FUNCTION_BLOCK "FB33 Ausgaege an FG"	// FB 33
TITLE = Ausgänge für Farbgrafik in Datenworte des DB33 speichern
//Erstellung:
//Datum        Bearbeiter                                                 Version
//--------------------------------------------------------------------------------
//00.00.00     xxx                                                        01.00.00
//
//Änderungen:
//Nr. Datum    Bearb Beschreibung                                   Marke Version
//--------------------------------------------------------------------------------
//01  00.00.00                                                      (xxx) xx.xx.xx
//
//--------------------------------------------------------------------------------
//
//
AUTHOR : sra
FAMILY : SCADA
NAME : outputs
VERSION : 0.0
VAR
  output_0_0 : BOOL ;
  output_0_1 : BOOL ;
  output_0_2 : BOOL ;
  output_0_3 : BOOL ;
  output_0_4 : BOOL ;
  output_0_5 : BOOL ;
  output_0_6 : BOOL ;
  output_0_7 : BOOL ;
  output_1_0 : BOOL ;
  output_1_1 : BOOL ;
  output_1_2 : BOOL ;
  output_1_3 : BOOL ;
  output_1_4 : BOOL ;
  output_1_5 : BOOL ;
  output_1_6 : BOOL ;
  output_1_7 : BOOL ;
  output_2_0 : BOOL ;
  output_2_1 : BOOL ;
  output_2_2 : BOOL ;
  output_2_3 : BOOL ;
  output_2_4 : BOOL ;
  output_2_5 : BOOL ;
  output_2_6 : BOOL ;
  output_2_7 : BOOL ;
  output_3_0 : BOOL ;
  output_3_1 : BOOL ;
  output_3_2 : BOOL ;
  output_3_3 : BOOL ;
  output_3_4 : BOOL ;
  output_3_5 : BOOL ;
  output_3_6 : BOOL ;
  output_3_7 : BOOL ;
  output_4_0 : BOOL ;
  output_4_1 : BOOL ;
  output_4_2 : BOOL ;
  output_4_3 : BOOL ;
  output_4_4 : BOOL ;
  output_4_5 : BOOL ;
  output_4_6 : BOOL ;
  output_4_7 : BOOL ;
  output_5_0 : BOOL ;
  output_5_1 : BOOL ;
  output_5_2 : BOOL ;
  output_5_3 : BOOL ;
  output_5_4 : BOOL ;
  output_5_5 : BOOL ;
  output_5_6 : BOOL ;
  output_5_7 : BOOL ;
  output_6_0 : BOOL ;
  output_6_1 : BOOL ;
  output_6_2 : BOOL ;
  output_6_3 : BOOL ;
  output_6_4 : BOOL ;
  output_6_5 : BOOL ;
  output_6_6 : BOOL ;
  output_6_7 : BOOL ;
  output_7_0 : BOOL ;
  output_7_1 : BOOL ;
  output_7_2 : BOOL ;
  output_7_3 : BOOL ;
  output_7_4 : BOOL ;
  output_7_5 : BOOL ;
  output_7_6 : BOOL ;
  output_7_7 : BOOL ;
  output_8_0 : BOOL ;
  output_8_1 : BOOL ;
  output_8_2 : BOOL ;
  output_8_3 : BOOL ;
  output_8_4 : BOOL ;
  output_8_5 : BOOL ;
  output_8_6 : BOOL ;
  output_8_7 : BOOL ;
  output_9_0 : BOOL ;
  output_9_1 : BOOL ;
  output_9_2 : BOOL ;
  output_9_3 : BOOL ;
  output_9_4 : BOOL ;
  output_9_5 : BOOL ;
  output_9_6 : BOOL ;
  output_9_7 : BOOL ;
  output_10_0 : BOOL ;
  output_10_1 : BOOL ;
  output_10_2 : BOOL ;
  output_10_3 : BOOL ;
  output_10_4 : BOOL ;
  output_10_5 : BOOL ;
  output_10_6 : BOOL ;
  output_10_7 : BOOL ;
  output_11_0 : BOOL ;
  output_11_1 : BOOL ;
  output_11_2 : BOOL ;
  output_11_3 : BOOL ;
  output_11_4 : BOOL ;
  output_11_5 : BOOL ;
  output_11_6 : BOOL ;
  output_11_7 : BOOL ;
  output_12_0 : BOOL ;
  output_12_1 : BOOL ;
  output_12_2 : BOOL ;
  output_12_3 : BOOL ;
  output_12_4 : BOOL ;
  output_12_5 : BOOL ;
  output_12_6 : BOOL ;
  output_12_7 : BOOL ;
  output_13_0 : BOOL ;
  output_13_1 : BOOL ;
  output_13_2 : BOOL ;
  output_13_3 : BOOL ;
  output_13_4 : BOOL ;
  output_13_5 : BOOL ;
  output_13_6 : BOOL ;
  output_13_7 : BOOL ;
  output_14_0 : BOOL ;
  output_14_1 : BOOL ;
  output_14_2 : BOOL ;
  output_14_3 : BOOL ;
  output_14_4 : BOOL ;
  output_14_5 : BOOL ;
  output_14_6 : BOOL ;
  output_14_7 : BOOL ;
  output_15_0 : BOOL ;
  output_15_1 : BOOL ;
  output_15_2 : BOOL ;
  output_15_3 : BOOL ;
  output_15_4 : BOOL ;
  output_15_5 : BOOL ;
  output_15_6 : BOOL ;
  output_15_7 : BOOL ;
  output_16_0 : BOOL ;
  output_16_1 : BOOL ;
  output_16_2 : BOOL ;
  output_16_3 : BOOL ;
  output_16_4 : BOOL ;
  output_16_5 : BOOL ;
  output_16_6 : BOOL ;
  output_16_7 : BOOL ;
  output_17_0 : BOOL ;
  output_17_1 : BOOL ;
  output_17_2 : BOOL ;
  output_17_3 : BOOL ;
  output_17_4 : BOOL ;
  output_17_5 : BOOL ;
  output_17_6 : BOOL ;
  output_17_7 : BOOL ;
  output_18_0 : BOOL ;
  output_18_1 : BOOL ;
  output_18_2 : BOOL ;
  output_18_3 : BOOL ;
  output_18_4 : BOOL ;
  output_18_5 : BOOL ;
  output_18_6 : BOOL ;
  output_18_7 : BOOL ;
  output_19_0 : BOOL ;
  output_19_1 : BOOL ;
  output_19_2 : BOOL ;
  output_19_3 : BOOL ;
  output_19_4 : BOOL ;
  output_19_5 : BOOL ;
  output_19_6 : BOOL ;
  output_19_7 : BOOL ;
  output_20_0 : BOOL ;
  output_20_1 : BOOL ;
  output_20_2 : BOOL ;
  output_20_3 : BOOL ;
  output_20_4 : BOOL ;
  output_20_5 : BOOL ;
  output_20_6 : BOOL ;
  output_20_7 : BOOL ;
  output_21_0 : BOOL ;
  output_21_1 : BOOL ;
  output_21_2 : BOOL ;
  output_21_3 : BOOL ;
  output_21_4 : BOOL ;
  output_21_5 : BOOL ;
  output_21_6 : BOOL ;
  output_21_7 : BOOL ;
  output_22_0 : BOOL ;
  output_22_1 : BOOL ;
  output_22_2 : BOOL ;
  output_22_3 : BOOL ;
  output_22_4 : BOOL ;
  output_22_5 : BOOL ;
  output_22_6 : BOOL ;
  output_22_7 : BOOL ;
  output_23_0 : BOOL ;
  output_23_1 : BOOL ;
  output_23_2 : BOOL ;
  output_23_3 : BOOL ;
  output_23_4 : BOOL ;
  output_23_5 : BOOL ;
  output_23_6 : BOOL ;
  output_23_7 : BOOL ;
  output_24_0 : BOOL ;
  output_24_1 : BOOL ;
  output_24_2 : BOOL ;
  output_24_3 : BOOL ;
  output_24_4 : BOOL ;
  output_24_5 : BOOL ;
  output_24_6 : BOOL ;
  output_24_7 : BOOL ;
  output_25_0 : BOOL ;
  output_25_1 : BOOL ;
  output_25_2 : BOOL ;
  output_25_3 : BOOL ;
  output_25_4 : BOOL ;
  output_25_5 : BOOL ;
  output_25_6 : BOOL ;
  output_25_7 : BOOL ;
  output_26_0 : BOOL ;
  output_26_1 : BOOL ;
  output_26_2 : BOOL ;
  output_26_3 : BOOL ;
  output_26_4 : BOOL ;
  output_26_5 : BOOL ;
  output_26_6 : BOOL ;
  output_26_7 : BOOL ;
  output_27_0 : BOOL ;
  output_27_1 : BOOL ;
  output_27_2 : BOOL ;
  output_27_3 : BOOL ;
  output_27_4 : BOOL ;
  output_27_5 : BOOL ;
  output_27_6 : BOOL ;
  output_27_7 : BOOL ;
  output_28_0 : BOOL ;
  output_28_1 : BOOL ;
  output_28_2 : BOOL ;
  output_28_3 : BOOL ;
  output_28_4 : BOOL ;
  output_28_5 : BOOL ;
  output_28_6 : BOOL ;
  output_28_7 : BOOL ;
  output_29_0 : BOOL ;
  output_29_1 : BOOL ;
  output_29_2 : BOOL ;
  output_29_3 : BOOL ;
  output_29_4 : BOOL ;
  output_29_5 : BOOL ;
  output_29_6 : BOOL ;
  output_29_7 : BOOL ;
  output_30_0 : BOOL ;
  output_30_1 : BOOL ;
  output_30_2 : BOOL ;
  output_30_3 : BOOL ;
  output_30_4 : BOOL ;
  output_30_5 : BOOL ;
  output_30_6 : BOOL ;
  output_30_7 : BOOL ;
  output_31_0 : BOOL ;
  output_31_1 : BOOL ;
  output_31_2 : BOOL ;
  output_31_3 : BOOL ;
  output_31_4 : BOOL ;
  output_31_5 : BOOL ;
  output_31_6 : BOOL ;
  output_31_7 : BOOL ;
  output_32_0 : BOOL ;
  output_32_1 : BOOL ;
  output_32_2 : BOOL ;
  output_32_3 : BOOL ;
  output_32_4 : BOOL ;
  output_32_5 : BOOL ;
  output_32_6 : BOOL ;
  output_32_7 : BOOL ;
  output_33_0 : BOOL ;
  output_33_1 : BOOL ;
  output_33_2 : BOOL ;
  output_33_3 : BOOL ;
  output_33_4 : BOOL ;
  output_33_5 : BOOL ;
  output_33_6 : BOOL ;
  output_33_7 : BOOL ;
  output_34_0 : BOOL ;
  output_34_1 : BOOL ;
  output_34_2 : BOOL ;
  output_34_3 : BOOL ;
  output_34_4 : BOOL ;
  output_34_5 : BOOL ;
  output_34_6 : BOOL ;
  output_34_7 : BOOL ;
  output_35_0 : BOOL ;
  output_35_1 : BOOL ;
  output_35_2 : BOOL ;
  output_35_3 : BOOL ;
  output_35_4 : BOOL ;
  output_35_5 : BOOL ;
  output_35_6 : BOOL ;
  output_35_7 : BOOL ;
  output_36_0 : BOOL ;
  output_36_1 : BOOL ;
  output_36_2 : BOOL ;
  output_36_3 : BOOL ;
  output_36_4 : BOOL ;
  output_36_5 : BOOL ;
  output_36_6 : BOOL ;
  output_36_7 : BOOL ;
  output_37_0 : BOOL ;
  output_37_1 : BOOL ;
  output_37_2 : BOOL ;
  output_37_3 : BOOL ;
  output_37_4 : BOOL ;
  output_37_5 : BOOL ;
  output_37_6 : BOOL ;
  output_37_7 : BOOL ;
  output_38_0 : BOOL ;
  output_38_1 : BOOL ;
  output_38_2 : BOOL ;
  output_38_3 : BOOL ;
  output_38_4 : BOOL ;
  output_38_5 : BOOL ;
  output_38_6 : BOOL ;
  output_38_7 : BOOL ;
  output_39_0 : BOOL ;
  output_39_1 : BOOL ;
  output_39_2 : BOOL ;
  output_39_3 : BOOL ;
  output_39_4 : BOOL ;
  output_39_5 : BOOL ;
  output_39_6 : BOOL ;
  output_39_7 : BOOL ;
  output_40_0 : BOOL ;
  output_40_1 : BOOL ;
  output_40_2 : BOOL ;
  output_40_3 : BOOL ;
  output_40_4 : BOOL ;
  output_40_5 : BOOL ;
  output_40_6 : BOOL ;
  output_40_7 : BOOL ;
  output_41_0 : BOOL ;
  output_41_1 : BOOL ;
  output_41_2 : BOOL ;
  output_41_3 : BOOL ;
  output_41_4 : BOOL ;
  output_41_5 : BOOL ;
  output_41_6 : BOOL ;
  output_41_7 : BOOL ;
  output_42_0 : BOOL ;
  output_42_1 : BOOL ;
  output_42_2 : BOOL ;
  output_42_3 : BOOL ;
  output_42_4 : BOOL ;
  output_42_5 : BOOL ;
  output_42_6 : BOOL ;
  output_42_7 : BOOL ;
  output_43_0 : BOOL ;
  output_43_1 : BOOL ;
  output_43_2 : BOOL ;
  output_43_3 : BOOL ;
  output_43_4 : BOOL ;
  output_43_5 : BOOL ;
  output_43_6 : BOOL ;
  output_43_7 : BOOL ;
  output_44_0 : BOOL ;
  output_44_1 : BOOL ;
  output_44_2 : BOOL ;
  output_44_3 : BOOL ;
  output_44_4 : BOOL ;
  output_44_5 : BOOL ;
  output_44_6 : BOOL ;
  output_44_7 : BOOL ;
  output_45_0 : BOOL ;
  output_45_1 : BOOL ;
  output_45_2 : BOOL ;
  output_45_3 : BOOL ;
  output_45_4 : BOOL ;
  output_45_5 : BOOL ;
  output_45_6 : BOOL ;
  output_45_7 : BOOL ;
  output_46_0 : BOOL ;
  output_46_1 : BOOL ;
  output_46_2 : BOOL ;
  output_46_3 : BOOL ;
  output_46_4 : BOOL ;
  output_46_5 : BOOL ;
  output_46_6 : BOOL ;
  output_46_7 : BOOL ;
  output_47_0 : BOOL ;
  output_47_1 : BOOL ;
  output_47_2 : BOOL ;
  output_47_3 : BOOL ;
  output_47_4 : BOOL ;
  output_47_5 : BOOL ;
  output_47_6 : BOOL ;
  output_47_7 : BOOL ;
  output_48_0 : BOOL ;
  output_48_1 : BOOL ;
  output_48_2 : BOOL ;
  output_48_3 : BOOL ;
  output_48_4 : BOOL ;
  output_48_5 : BOOL ;
  output_48_6 : BOOL ;
  output_48_7 : BOOL ;
  output_49_0 : BOOL ;
  output_49_1 : BOOL ;
  output_49_2 : BOOL ;
  output_49_3 : BOOL ;
  output_49_4 : BOOL ;
  output_49_5 : BOOL ;
  output_49_6 : BOOL ;
  output_49_7 : BOOL ;
  output_50_0 : BOOL ;
  output_50_1 : BOOL ;
  output_50_2 : BOOL ;
  output_50_3 : BOOL ;
  output_50_4 : BOOL ;
  output_50_5 : BOOL ;
  output_50_6 : BOOL ;
  output_50_7 : BOOL ;
  output_51_0 : BOOL ;
  output_51_1 : BOOL ;
  output_51_2 : BOOL ;
  output_51_3 : BOOL ;
  output_51_4 : BOOL ;
  output_51_5 : BOOL ;
  output_51_6 : BOOL ;
  output_51_7 : BOOL ;
  output_52_0 : BOOL ;
  output_52_1 : BOOL ;
  output_52_2 : BOOL ;
  output_52_3 : BOOL ;
  output_52_4 : BOOL ;
  output_52_5 : BOOL ;
  output_52_6 : BOOL ;
  output_52_7 : BOOL ;
  output_53_0 : BOOL ;
  output_53_1 : BOOL ;
  output_53_2 : BOOL ;
  output_53_3 : BOOL ;
  output_53_4 : BOOL ;
  output_53_5 : BOOL ;
  output_53_6 : BOOL ;
  output_53_7 : BOOL ;
  output_54_0 : BOOL ;
  output_54_1 : BOOL ;
  output_54_2 : BOOL ;
  output_54_3 : BOOL ;
  output_54_4 : BOOL ;
  output_54_5 : BOOL ;
  output_54_6 : BOOL ;
  output_54_7 : BOOL ;
  output_55_0 : BOOL ;
  output_55_1 : BOOL ;
  output_55_2 : BOOL ;
  output_55_3 : BOOL ;
  output_55_4 : BOOL ;
  output_55_5 : BOOL ;
  output_55_6 : BOOL ;
  output_55_7 : BOOL ;
  output_56_0 : BOOL ;
  output_56_1 : BOOL ;
  output_56_2 : BOOL ;
  output_56_3 : BOOL ;
  output_56_4 : BOOL ;
  output_56_5 : BOOL ;
  output_56_6 : BOOL ;
  output_56_7 : BOOL ;
  output_57_0 : BOOL ;
  output_57_1 : BOOL ;
  output_57_2 : BOOL ;
  output_57_3 : BOOL ;
  output_57_4 : BOOL ;
  output_57_5 : BOOL ;
  output_57_6 : BOOL ;
  output_57_7 : BOOL ;
  output_58_0 : BOOL ;
  output_58_1 : BOOL ;
  output_58_2 : BOOL ;
  output_58_3 : BOOL ;
  output_58_4 : BOOL ;
  output_58_5 : BOOL ;
  output_58_6 : BOOL ;
  output_58_7 : BOOL ;
  output_59_0 : BOOL ;
  output_59_1 : BOOL ;
  output_59_2 : BOOL ;
  output_59_3 : BOOL ;
  output_59_4 : BOOL ;
  output_59_5 : BOOL ;
  output_59_6 : BOOL ;
  output_59_7 : BOOL ;
  output_60_0 : BOOL ;
  output_60_1 : BOOL ;
  output_60_2 : BOOL ;
  output_60_3 : BOOL ;
  output_60_4 : BOOL ;
  output_60_5 : BOOL ;
  output_60_6 : BOOL ;
  output_60_7 : BOOL ;
  output_61_0 : BOOL ;
  output_61_1 : BOOL ;
  output_61_2 : BOOL ;
  output_61_3 : BOOL ;
  output_61_4 : BOOL ;
  output_61_5 : BOOL ;
  output_61_6 : BOOL ;
  output_61_7 : BOOL ;
  output_62_0 : BOOL ;
  output_62_1 : BOOL ;
  output_62_2 : BOOL ;
  output_62_3 : BOOL ;
  output_62_4 : BOOL ;
  output_62_5 : BOOL ;
  output_62_6 : BOOL ;
  output_62_7 : BOOL ;
  output_63_0 : BOOL ;
  output_63_1 : BOOL ;
  output_63_2 : BOOL ;
  output_63_3 : BOOL ;
  output_63_4 : BOOL ;
  output_63_5 : BOOL ;
  output_63_6 : BOOL ;
  output_63_7 : BOOL ;
  output_64_0 : BOOL ;
  output_64_1 : BOOL ;
  output_64_2 : BOOL ;
  output_64_3 : BOOL ;
  output_64_4 : BOOL ;
  output_64_5 : BOOL ;
  output_64_6 : BOOL ;
  output_64_7 : BOOL ;
  output_65_0 : BOOL ;
  output_65_1 : BOOL ;
  output_65_2 : BOOL ;
  output_65_3 : BOOL ;
  output_65_4 : BOOL ;
  output_65_5 : BOOL ;
  output_65_6 : BOOL ;
  output_65_7 : BOOL ;
  output_66_0 : BOOL ;
  output_66_1 : BOOL ;
  output_66_2 : BOOL ;
  output_66_3 : BOOL ;
  output_66_4 : BOOL ;
  output_66_5 : BOOL ;
  output_66_6 : BOOL ;
  output_66_7 : BOOL ;
  output_67_0 : BOOL ;
  output_67_1 : BOOL ;
  output_67_2 : BOOL ;
  output_67_3 : BOOL ;
  output_67_4 : BOOL ;
  output_67_5 : BOOL ;
  output_67_6 : BOOL ;
  output_67_7 : BOOL ;
  output_68_0 : BOOL ;
  output_68_1 : BOOL ;
  output_68_2 : BOOL ;
  output_68_3 : BOOL ;
  output_68_4 : BOOL ;
  output_68_5 : BOOL ;
  output_68_6 : BOOL ;
  output_68_7 : BOOL ;
  output_69_0 : BOOL ;
  output_69_1 : BOOL ;
  output_69_2 : BOOL ;
  output_69_3 : BOOL ;
  output_69_4 : BOOL ;
  output_69_5 : BOOL ;
  output_69_6 : BOOL ;
  output_69_7 : BOOL ;
  output_70_0 : BOOL ;
  output_70_1 : BOOL ;
  output_70_2 : BOOL ;
  output_70_3 : BOOL ;
  output_70_4 : BOOL ;
  output_70_5 : BOOL ;
  output_70_6 : BOOL ;
  output_70_7 : BOOL ;
  output_71_0 : BOOL ;
  output_71_1 : BOOL ;
  output_71_2 : BOOL ;
  output_71_3 : BOOL ;
  output_71_4 : BOOL ;
  output_71_5 : BOOL ;
  output_71_6 : BOOL ;
  output_71_7 : BOOL ;
  output_72_0 : BOOL ;
  output_72_1 : BOOL ;
  output_72_2 : BOOL ;
  output_72_3 : BOOL ;
  output_72_4 : BOOL ;
  output_72_5 : BOOL ;
  output_72_6 : BOOL ;
  output_72_7 : BOOL ;
  output_73_0 : BOOL ;
  output_73_1 : BOOL ;
  output_73_2 : BOOL ;
  output_73_3 : BOOL ;
  output_73_4 : BOOL ;
  output_73_5 : BOOL ;
  output_73_6 : BOOL ;
  output_73_7 : BOOL ;
  output_74_0 : BOOL ;
  output_74_1 : BOOL ;
  output_74_2 : BOOL ;
  output_74_3 : BOOL ;
  output_74_4 : BOOL ;
  output_74_5 : BOOL ;
  output_74_6 : BOOL ;
  output_74_7 : BOOL ;
  output_75_0 : BOOL ;
  output_75_1 : BOOL ;
  output_75_2 : BOOL ;
  output_75_3 : BOOL ;
  output_75_4 : BOOL ;
  output_75_5 : BOOL ;
  output_75_6 : BOOL ;
  output_75_7 : BOOL ;
  output_76_0 : BOOL ;
  output_76_1 : BOOL ;
  output_76_2 : BOOL ;
  output_76_3 : BOOL ;
  output_76_4 : BOOL ;
  output_76_5 : BOOL ;
  output_76_6 : BOOL ;
  output_76_7 : BOOL ;
  output_77_0 : BOOL ;
  output_77_1 : BOOL ;
  output_77_2 : BOOL ;
  output_77_3 : BOOL ;
  output_77_4 : BOOL ;
  output_77_5 : BOOL ;
  output_77_6 : BOOL ;
  output_77_7 : BOOL ;
  output_78_0 : BOOL ;
  output_78_1 : BOOL ;
  output_78_2 : BOOL ;
  output_78_3 : BOOL ;
  output_78_4 : BOOL ;
  output_78_5 : BOOL ;
  output_78_6 : BOOL ;
  output_78_7 : BOOL ;
  output_79_0 : BOOL ;
  output_79_1 : BOOL ;
  output_79_2 : BOOL ;
  output_79_3 : BOOL ;
  output_79_4 : BOOL ;
  output_79_5 : BOOL ;
  output_79_6 : BOOL ;
  output_79_7 : BOOL ;
  output_80_0 : BOOL ;
  output_80_1 : BOOL ;
  output_80_2 : BOOL ;
  output_80_3 : BOOL ;
  output_80_4 : BOOL ;
  output_80_5 : BOOL ;
  output_80_6 : BOOL ;
  output_80_7 : BOOL ;
  output_81_0 : BOOL ;
  output_81_1 : BOOL ;
  output_81_2 : BOOL ;
  output_81_3 : BOOL ;
  output_81_4 : BOOL ;
  output_81_5 : BOOL ;
  output_81_6 : BOOL ;
  output_81_7 : BOOL ;
  output_82_0 : BOOL ;
  output_82_1 : BOOL ;
  output_82_2 : BOOL ;
  output_82_3 : BOOL ;
  output_82_4 : BOOL ;
  output_82_5 : BOOL ;
  output_82_6 : BOOL ;
  output_82_7 : BOOL ;
  output_83_0 : BOOL ;
  output_83_1 : BOOL ;
  output_83_2 : BOOL ;
  output_83_3 : BOOL ;
  output_83_4 : BOOL ;
  output_83_5 : BOOL ;
  output_83_6 : BOOL ;
  output_83_7 : BOOL ;
  output_84_0 : BOOL ;
  output_84_1 : BOOL ;
  output_84_2 : BOOL ;
  output_84_3 : BOOL ;
  output_84_4 : BOOL ;
  output_84_5 : BOOL ;
  output_84_6 : BOOL ;
  output_84_7 : BOOL ;
  output_85_0 : BOOL ;
  output_85_1 : BOOL ;
  output_85_2 : BOOL ;
  output_85_3 : BOOL ;
  output_85_4 : BOOL ;
  output_85_5 : BOOL ;
  output_85_6 : BOOL ;
  output_85_7 : BOOL ;
  output_86_0 : BOOL ;
  output_86_1 : BOOL ;
  output_86_2 : BOOL ;
  output_86_3 : BOOL ;
  output_86_4 : BOOL ;
  output_86_5 : BOOL ;
  output_86_6 : BOOL ;
  output_86_7 : BOOL ;
  output_87_0 : BOOL ;
  output_87_1 : BOOL ;
  output_87_2 : BOOL ;
  output_87_3 : BOOL ;
  output_87_4 : BOOL ;
  output_87_5 : BOOL ;
  output_87_6 : BOOL ;
  output_87_7 : BOOL ;
  output_88_0 : BOOL ;
  output_88_1 : BOOL ;
  output_88_2 : BOOL ;
  output_88_3 : BOOL ;
  output_88_4 : BOOL ;
  output_88_5 : BOOL ;
  output_88_6 : BOOL ;
  output_88_7 : BOOL ;
  output_89_0 : BOOL ;
  output_89_1 : BOOL ;
  output_89_2 : BOOL ;
  output_89_3 : BOOL ;
  output_89_4 : BOOL ;
  output_89_5 : BOOL ;
  output_89_6 : BOOL ;
  output_89_7 : BOOL ;
  output_90_0 : BOOL ;
  output_90_1 : BOOL ;
  output_90_2 : BOOL ;
  output_90_3 : BOOL ;
  output_90_4 : BOOL ;
  output_90_5 : BOOL ;
  output_90_6 : BOOL ;
  output_90_7 : BOOL ;
  output_91_0 : BOOL ;
  output_91_1 : BOOL ;
  output_91_2 : BOOL ;
  output_91_3 : BOOL ;
  output_91_4 : BOOL ;
  output_91_5 : BOOL ;
  output_91_6 : BOOL ;
  output_91_7 : BOOL ;
  output_92_0 : BOOL ;
  output_92_1 : BOOL ;
  output_92_2 : BOOL ;
  output_92_3 : BOOL ;
  output_92_4 : BOOL ;
  output_92_5 : BOOL ;
  output_92_6 : BOOL ;
  output_92_7 : BOOL ;
  output_93_0 : BOOL ;
  output_93_1 : BOOL ;
  output_93_2 : BOOL ;
  output_93_3 : BOOL ;
  output_93_4 : BOOL ;
  output_93_5 : BOOL ;
  output_93_6 : BOOL ;
  output_93_7 : BOOL ;
  output_94_0 : BOOL ;
  output_94_1 : BOOL ;
  output_94_2 : BOOL ;
  output_94_3 : BOOL ;
  output_94_4 : BOOL ;
  output_94_5 : BOOL ;
  output_94_6 : BOOL ;
  output_94_7 : BOOL ;
  output_95_0 : BOOL ;
  output_95_1 : BOOL ;
  output_95_2 : BOOL ;
  output_95_3 : BOOL ;
  output_95_4 : BOOL ;
  output_95_5 : BOOL ;
  output_95_6 : BOOL ;
  output_95_7 : BOOL ;
  output_96_0 : BOOL ;
  output_96_1 : BOOL ;
  output_96_2 : BOOL ;
  output_96_3 : BOOL ;
  output_96_4 : BOOL ;
  output_96_5 : BOOL ;
  output_96_6 : BOOL ;
  output_96_7 : BOOL ;
  output_97_0 : BOOL ;
  output_97_1 : BOOL ;
  output_97_2 : BOOL ;
  output_97_3 : BOOL ;
  output_97_4 : BOOL ;
  output_97_5 : BOOL ;
  output_97_6 : BOOL ;
  output_97_7 : BOOL ;
  output_98_0 : BOOL ;
  output_98_1 : BOOL ;
  output_98_2 : BOOL ;
  output_98_3 : BOOL ;
  output_98_4 : BOOL ;
  output_98_5 : BOOL ;
  output_98_6 : BOOL ;
  output_98_7 : BOOL ;
  output_99_0 : BOOL ;
  output_99_1 : BOOL ;
  output_99_2 : BOOL ;
  output_99_3 : BOOL ;
  output_99_4 : BOOL ;
  output_99_5 : BOOL ;
  output_99_6 : BOOL ;
  output_99_7 : BOOL ;
  output_100_0 : BOOL ;
  output_100_1 : BOOL ;
  output_100_2 : BOOL ;
  output_100_3 : BOOL ;
  output_100_4 : BOOL ;
  output_100_5 : BOOL ;
  output_100_6 : BOOL ;
  output_100_7 : BOOL ;
  output_101_0 : BOOL ;
  output_101_1 : BOOL ;
  output_101_2 : BOOL ;
  output_101_3 : BOOL ;
  output_101_4 : BOOL ;
  output_101_5 : BOOL ;
  output_101_6 : BOOL ;
  output_101_7 : BOOL ;
  output_102_0 : BOOL ;
  output_102_1 : BOOL ;
  output_102_2 : BOOL ;
  output_102_3 : BOOL ;
  output_102_4 : BOOL ;
  output_102_5 : BOOL ;
  output_102_6 : BOOL ;
  output_102_7 : BOOL ;
  output_103_0 : BOOL ;
  output_103_1 : BOOL ;
  output_103_2 : BOOL ;
  output_103_3 : BOOL ;
  output_103_4 : BOOL ;
  output_103_5 : BOOL ;
  output_103_6 : BOOL ;
  output_103_7 : BOOL ;
  output_104_0 : BOOL ;
  output_104_1 : BOOL ;
  output_104_2 : BOOL ;
  output_104_3 : BOOL ;
  output_104_4 : BOOL ;
  output_104_5 : BOOL ;
  output_104_6 : BOOL ;
  output_104_7 : BOOL ;
  output_105_0 : BOOL ;
  output_105_1 : BOOL ;
  output_105_2 : BOOL ;
  output_105_3 : BOOL ;
  output_105_4 : BOOL ;
  output_105_5 : BOOL ;
  output_105_6 : BOOL ;
  output_105_7 : BOOL ;
  output_106_0 : BOOL ;
  output_106_1 : BOOL ;
  output_106_2 : BOOL ;
  output_106_3 : BOOL ;
  output_106_4 : BOOL ;
  output_106_5 : BOOL ;
  output_106_6 : BOOL ;
  output_106_7 : BOOL ;
  output_107_0 : BOOL ;
  output_107_1 : BOOL ;
  output_107_2 : BOOL ;
  output_107_3 : BOOL ;
  output_107_4 : BOOL ;
  output_107_5 : BOOL ;
  output_107_6 : BOOL ;
  output_107_7 : BOOL ;
  output_108_0 : BOOL ;
  output_108_1 : BOOL ;
  output_108_2 : BOOL ;
  output_108_3 : BOOL ;
  output_108_4 : BOOL ;
  output_108_5 : BOOL ;
  output_108_6 : BOOL ;
  output_108_7 : BOOL ;
  output_109_0 : BOOL ;
  output_109_1 : BOOL ;
  output_109_2 : BOOL ;
  output_109_3 : BOOL ;
  output_109_4 : BOOL ;
  output_109_5 : BOOL ;
  output_109_6 : BOOL ;
  output_109_7 : BOOL ;
  output_110_0 : BOOL ;
  output_110_1 : BOOL ;
  output_110_2 : BOOL ;
  output_110_3 : BOOL ;
  output_110_4 : BOOL ;
  output_110_5 : BOOL ;
  output_110_6 : BOOL ;
  output_110_7 : BOOL ;
  output_111_0 : BOOL ;
  output_111_1 : BOOL ;
  output_111_2 : BOOL ;
  output_111_3 : BOOL ;
  output_111_4 : BOOL ;
  output_111_5 : BOOL ;
  output_111_6 : BOOL ;
  output_111_7 : BOOL ;
  output_112_0 : BOOL ;
  output_112_1 : BOOL ;
  output_112_2 : BOOL ;
  output_112_3 : BOOL ;
  output_112_4 : BOOL ;
  output_112_5 : BOOL ;
  output_112_6 : BOOL ;
  output_112_7 : BOOL ;
  output_113_0 : BOOL ;
  output_113_1 : BOOL ;
  output_113_2 : BOOL ;
  output_113_3 : BOOL ;
  output_113_4 : BOOL ;
  output_113_5 : BOOL ;
  output_113_6 : BOOL ;
  output_113_7 : BOOL ;
  output_114_0 : BOOL ;
  output_114_1 : BOOL ;
  output_114_2 : BOOL ;
  output_114_3 : BOOL ;
  output_114_4 : BOOL ;
  output_114_5 : BOOL ;
  output_114_6 : BOOL ;
  output_114_7 : BOOL ;
  output_115_0 : BOOL ;
  output_115_1 : BOOL ;
  output_115_2 : BOOL ;
  output_115_3 : BOOL ;
  output_115_4 : BOOL ;
  output_115_5 : BOOL ;
  output_115_6 : BOOL ;
  output_115_7 : BOOL ;
  output_116_0 : BOOL ;
  output_116_1 : BOOL ;
  output_116_2 : BOOL ;
  output_116_3 : BOOL ;
  output_116_4 : BOOL ;
  output_116_5 : BOOL ;
  output_116_6 : BOOL ;
  output_116_7 : BOOL ;
  output_117_0 : BOOL ;
  output_117_1 : BOOL ;
  output_117_2 : BOOL ;
  output_117_3 : BOOL ;
  output_117_4 : BOOL ;
  output_117_5 : BOOL ;
  output_117_6 : BOOL ;
  output_117_7 : BOOL ;
  output_118_0 : BOOL ;
  output_118_1 : BOOL ;
  output_118_2 : BOOL ;
  output_118_3 : BOOL ;
  output_118_4 : BOOL ;
  output_118_5 : BOOL ;
  output_118_6 : BOOL ;
  output_118_7 : BOOL ;
  output_119_0 : BOOL ;
  output_119_1 : BOOL ;
  output_119_2 : BOOL ;
  output_119_3 : BOOL ;
  output_119_4 : BOOL ;
  output_119_5 : BOOL ;
  output_119_6 : BOOL ;
  output_119_7 : BOOL ;
  output_120_0 : BOOL ;
  output_120_1 : BOOL ;
  output_120_2 : BOOL ;
  output_120_3 : BOOL ;
  output_120_4 : BOOL ;
  output_120_5 : BOOL ;
  output_120_6 : BOOL ;
  output_120_7 : BOOL ;
  output_121_0 : BOOL ;
  output_121_1 : BOOL ;
  output_121_2 : BOOL ;
  output_121_3 : BOOL ;
  output_121_4 : BOOL ;
  output_121_5 : BOOL ;
  output_121_6 : BOOL ;
  output_121_7 : BOOL ;
  output_122_0 : BOOL ;
  output_122_1 : BOOL ;
  output_122_2 : BOOL ;
  output_122_3 : BOOL ;
  output_122_4 : BOOL ;
  output_122_5 : BOOL ;
  output_122_6 : BOOL ;
  output_122_7 : BOOL ;
  output_123_0 : BOOL ;
  output_123_1 : BOOL ;
  output_123_2 : BOOL ;
  output_123_3 : BOOL ;
  output_123_4 : BOOL ;
  output_123_5 : BOOL ;
  output_123_6 : BOOL ;
  output_123_7 : BOOL ;
  output_124_0 : BOOL ;
  output_124_1 : BOOL ;
  output_124_2 : BOOL ;
  output_124_3 : BOOL ;
  output_124_4 : BOOL ;
  output_124_5 : BOOL ;
  output_124_6 : BOOL ;
  output_124_7 : BOOL ;
  output_125_0 : BOOL ;
  output_125_1 : BOOL ;
  output_125_2 : BOOL ;
  output_125_3 : BOOL ;
  output_125_4 : BOOL ;
  output_125_5 : BOOL ;
  output_125_6 : BOOL ;
  output_125_7 : BOOL ;
  output_126_0 : BOOL ;
  output_126_1 : BOOL ;
  output_126_2 : BOOL ;
  output_126_3 : BOOL ;
  output_126_4 : BOOL ;
  output_126_5 : BOOL ;
  output_126_6 : BOOL ;
  output_126_7 : BOOL ;
  output_127_0 : BOOL ;
  output_127_1 : BOOL ;
  output_127_2 : BOOL ;
  output_127_3 : BOOL ;
  output_127_4 : BOOL ;
  output_127_5 : BOOL ;
  output_127_6 : BOOL ;
  output_127_7 : BOOL ;
  output_128_0 : BOOL ;
  output_128_1 : BOOL ;
  output_128_2 : BOOL ;
  output_128_3 : BOOL ;
  output_128_4 : BOOL ;
  output_128_5 : BOOL ;
  output_128_6 : BOOL ;
  output_128_7 : BOOL ;
  output_129_0 : BOOL ;
  output_129_1 : BOOL ;
  output_129_2 : BOOL ;
  output_129_3 : BOOL ;
  output_129_4 : BOOL ;
  output_129_5 : BOOL ;
  output_129_6 : BOOL ;
  output_129_7 : BOOL ;
  reserve : ARRAY  [130 .. 1000 ] OF BYTE ;
END_VAR
BEGIN
NETWORK
TITLE = UR1
//!!!!! Beispiel !!!!!  
//
      L     QW 4;
      T     DIW 4;
      L     QW 8;
      T     DIW 8;
      L     QW 12;
      T     DIW 12;
      L     QW 16;
      T     DIW 16;
      L     QW 20;
      T     DIW 20;
      L     QW 24;
      T     DIW 24;
      L     QW 28;
      T     DIW 28;
NETWORK
TITLE = ET200B Module
//!!!!! Beispiel !!!!!  
//
//      L     QD    56
//      T     DID   56
//      L     QD    60
//      T     DID   60
//      L     QD    64
//      T     DID   64
//      L     QD    68
//      T     DID   68
//      L     QD    72
//      T     DID   72
//      L     QD    76
//      T     DID   76
//      L     QD    80
//      T     DID   80
//      L     QD    84
//      T     DID   84
END_FUNCTION_BLOCK

FUNCTION_BLOCK "FB34 Störbearbeitung"	// FB 34
TITLE = Störauswertung
//Erstellung:
//Datum        Bearbeiter                                                 Version
//--------------------------------------------------------------------------------
//
//
//Änderungen:
//Nr. Datum    Bearb Änderung                                       Marke  Version
//--------------------------------------------------------------------------------
// 
AUTHOR : sra
FAMILY : AZO
VERSION : 0.0
VAR
  Stoerung_E : ARRAY  [0 .. 255, 0 .. 7 ] OF BOOL ;
  Erstwertmeldung_E : ARRAY  [0 .. 255, 0 .. 7 ] OF BOOL ;
  Spiegelung_PC_Fehler_E : ARRAY  [0 .. 255, 0 .. 7 ] OF BOOL ;
  Quittierung_von_PC_E : ARRAY  [0 .. 255, 0 .. 7 ] OF BOOL ;
  Quittierung_von_OP : ARRAY  [0 .. 255, 0 .. 7 ] OF //acknowledge bits from Siemens panel
  BOOL ;
  alte_Quittieung_von_OP : ARRAY  [0 .. 255, 0 .. 7 ] OF //acknowledge bits from Siemens panel one cycle before
  BOOL ;
END_VAR
VAR_TEMP
  Ack_Fault : BOOL ;
END_VAR
BEGIN
NETWORK
TITLE = CPU Fehler
      L     DB3.DBW 30;
      T     DB34.DBW 0;
NETWORK
TITLE = Erstwertmeldung / Quittierung
      CALL  "FC16 Störauswertung" (
           Conf_AckBySiemensOP      := TRUE,
           Stoerungstakt            := "M4.7 ImpulseClock2,0Sec",
           Freigabe_Sammelstoerung  := FALSE,
           Quittierung              := #Ack_Fault,
           Stoerungs_DB             := 34,
           Quittierungs_DB_SCADA    := 35,
           Anzahl_Stoerungs_Byte    := 256,
           Offset_Stoerungs_Byte    := 0,
           Adresse_Anfangswort      := 0,
           Bereichslaenge           := 256,
           Sammelstoerung           := "M1.1 Fault(General)",
           Erstmeldung              := "M1.2 NewFault(General)",
           Erstmeldung_PC           := M 8.0,
           Quittierung_PC           := M 8.1);
NETWORK
TITLE = CPU Fehler löschen
      L     DB3.DBW 30;
      L     DB35.DBW 0;
      INVI;
      AW;
      T     DB3.DBW 30;
END_FUNCTION_BLOCK

FUNCTION_BLOCK "FB92 Eingänge AVP"	// FB 92
TITLE = Analogeingänge
//Erstellung:
//Datum        Bearbeiter                                                 Version
//--------------------------------------------------------------------------------
//??.??.??     M.Böhrer (bms)                                            01.00.00
//
//Änderungen:
//Nr. Datum    Bearbeiter         Änderung                                Version
//--------------------------------------------------------------------------------
//01  25.10.07 bms   Erweiterung AH200098L-N ..................... (001) 01.01.00 
//________________________________________________________________________________
//Funktion:
VERSION : 0.1
VAR
  Reserve : ARRAY  [0 .. 119 ] OF //(001)
  BYTE ;
  Drucktransmitter_VP09 : WORD ;	//(001)
  Drucktransmitter_VP10 : WORD ;	//(001)
  Drucktransmitter_VP16 : WORD ;	//(001)
  Drucktransmitter_VP17 : WORD ;	//(001)
  Drucktransmitter_VP20 : WORD ;
  Drucktransmitter_VP00 : WORD ;
  Drucktransmitter_VP08 : WORD ;
  Drucktransmitter_VP07 : WORD ;
  Eingang_analog_res_1 : ARRAY  [136 .. 142 ] OF BYTE ;
  Drucktransmitter_VP14 : WORD ;	//(001)
  Drucktransmitter_VP15 : WORD ;	//(001)
  Drucktransmitter_VP02 : WORD ;	//(001)
  Drucktransmitter_VP03 : WORD ;	//(001)
  Drucktransmitter_VP04 : WORD ;	//(001)
  Drucktransmitter_VP05 : WORD ;	//(001)
  Drucktransmitter_VP06 : WORD ;	//(001)
  Drucktransmitter_VPxx : WORD ;
  Wiegezelle_Silo_S_1 : WORD ;
  Wiegezelle_Silo_S_2 : WORD ;
  Wiegezelle_Silo_S_3 : WORD ;
  Wiegezelle_Silo_S_4 : WORD ;
  Wiegezelle_Silo_S_5 : WORD ;
  Eingang_analog_res_2 : ARRAY  [170 .. 398 ] OF BYTE ;
  Drucktransmitter_VPxxx : WORD ;
  Eingang_analog_res_3 : ARRAY  [408 .. 1022 ] OF BYTE ;
END_VAR
BEGIN
NETWORK
TITLE =
      BEU;
END_FUNCTION_BLOCK

FUNCTION_BLOCK "****PRODUCTION****"	// FB 1000
TITLE = Call Production FB's
//Creation:
//Date:            Author:                                               Version
//-------------------------------------------------------------------------------
//10.10.19     Ilia Bedniakov(ilia)                                      01.00.00
//
//Changes:
//No. Date:        Who       Description                           Mark   Version 
//-------------------------------------------------------------------------------
//-
//01
//_______________________________________________________________________________
//_
//Function:
AUTHOR : ilia
NAME : project
VERSION : 0.1
VAR_TEMP
  dummy_bool : BOOL ;
  conditionAcoustic : BOOL ;
END_VAR
BEGIN
NETWORK
TITLE = CALL RECEIVER REC01
      CALL  "RECEIVER" , "RECEIVER REC01" (
           I_iIFVacuumPumpDB        := 1051,
           I_iIFVacuumPumpDW        := 1051,
           I_iIFStorageDB           := 1001,
           I_iIFStorageDW           := 1001,
           I_iIFStoLocParDB         := 1001,
           I_xSystemActive          := DB30.DBX 102.0,
           I_xAngleValveOpen        := "02_02_101_Gp",
           I_xAngleValveClose       := "02_02_101_Gn",
           i_xPendelFlapREC         := "02_02_602_Gn",
           i_xHighLevelREC          := "02_02_601_Lp",
           I_xPFC_PM1               := "02_03_601_ES",
           I_xPFC_PM2               := "02_03_602_ES",
           i_xAckFullReceiver       := "DB35 Acknolegments".Quittierung[6, 0],
           i_xAngleValve            := "DB35 Acknolegments".Quittierung[4, 3],
           q_xAngleValve            := "02_02_101_UVp",
           q_xCleaningValve         := "02_02_102_UVp",
           q_xRepperValve           := "02_02_103_UVp",
           q_xRedLamp               := "10_01_501_H",
           q_xYellowLamp            := "10_01_502_H",
           q_xGreenLamp             := "10_01_503_H",
           f_xAngleValve            := DB34.DBX 4.3,
           f_xFullReceiver          := DB34.DBX 6.0,
           f_xNoStartConditions     := DB34.DBX 400.0,
           f_xNoPFCRequest          := DB34.DBX 400.1);
NETWORK
TITLE = CALL FAULTS AND CONTAINERSTATION CST01
      A     DB34.DBX 8.5;
      AN    "DB35 Acknolegments".Quittierung[8, 5];
      O;
      A     DB34.DBX 202.3;
      AN    "DB35 Acknolegments".Quittierung[202, 3];
      =     #conditionAcoustic;
      CALL  "CONTAINERSTATION" , "CONTAINERSTATION CST01" (
           i_xSystemActive          := DB30.DBX 102.0,
           i_xFAValveOpen           := "01_01_101_Gp",
           i_xFAValveClosed         := "01_01_101_Gn",
           i_xPBStart               := "01_01_601_H",
           i_xPBStop                := "01_01_602_H",
           i_xCstAvalible           := "01_01_603_H",
           ack_FAValve              := "DB35 Acknolegments".Quittierung[4, 7],
           q_xFAValve               := "01_01_101_UVp",
           q_xPFCMix                := "Q 10.2",
           q_xLMStart               := "01_01_501_H",
           q_xLMCstAvalible         := "01_01_502_H",
           f_xFAValve               := DB34.DBX 4.7);
NETWORK
TITLE = CALL  VACUUM PUMP PMP01
      CALL  "VACUUM PUMP" , "VP01" (
           IF_VP1_FC_DB             := 1051,
           IF_VP1_FC_DW             := 1051,
           i_piwPressureVP1         := IW 200,
           i_xFAValveClose          := "02_01_101_Gn",
           i_xFAValveOpen           := "02_01_101_Gp",
           i_xSystemActive          := DB30.DBX 102.0,
           ack_xFAValve             := "DB35 Acknolegments".Quittierung[4, 1],
           ack_OverPressureVP1      := "DB35 Acknolegments".Quittierung[200, 0],
           q_xFAValve               := "02_01_101_UVn",
           f_xFAValve               := DB34.DBX 4.1,
           f_xPressureFaultVP1      := DB34.DBX 200.0,
           f_xBrokenWirePTVPV1      := DB34.DBX 200.1,
           f_xParErrorPTVPVP1       := DB34.DBX 200.2);
NETWORK
TITLE = CALL  FREQUENCY CONVERTERS (FC01)
      CALL  "*** FCs ***" , "FREQUENCY CONVERTERS";
END_FUNCTION_BLOCK

FUNCTION_BLOCK "CONTAINERSTATION"	// FB 1001
TITLE = HOPPER
//Creation:
//Date:            Author:                                               Version
//--------------------------------------------------------------------------------
//17.04.17          Ilia Bedniakov (ilia   )                             01.00.00
//
//Changes:
//No. Date:        Who       Description                           Mark   Version 
//--------------------------------------------------------------------------------
//01  17.07.2017   ilia      correction at comissioning            (001)  01.01.00
//02  19.07.2017   ilia     correction at comission                (002)  01.02.00
//03  19.10.2017   ilia     hopper emptying                        (003)  01.03.00
//04  02.08.2018   ilia     changing for project                
//________________________________________________________________________________
//Function:
AUTHOR : ilia
NAME : project
VERSION : 0.1
VAR_INPUT
  i_xSystemActive : BOOL ;	//system control on
  i_xFAValveOpen : BOOL ;
  i_xFAValveClosed : BOOL ;
  i_xPBStart : BOOL ;	//Start Button
  i_xPBStop : BOOL ;	//StopButton
  i_xCstAvalible : BOOL ;	//Container On Place
  ack_FAValve : BOOL ;	//acknowlege FAValve
END_VAR
VAR_IN_OUT
  q_xFAValve : BOOL ;	//Open Fresh Air Valve
  q_xPFCMix : BOOL ;	//Container in position PFC to MIX01
  q_xLMStart : BOOL ;
  q_xLMCstAvalible : BOOL ;
  f_xFAValve : BOOL ;	//feedback fault
END_VAR
VAR
  reserve_IO : ARRAY  [4 .. 49 ] OF BYTE ;
  HMI : STRUCT 	//Interface of HMI
   CMD : STRUCT
    xxRelease : BOOL ;
    SetEmpty : BOOL ;
    StopProd : BOOL ;
    StartProd : BOOL ;
    reserve_5 : BOOL ;
    reserve_6 : BOOL ;
    reserve_7 : BOOL ;
    reserve_8 : BOOL ;
    reserve_9 : BOOL ;
    reserve_10 : BOOL ;
    reserve_11 : BOOL ;
    reserve_12 : BOOL ;
    reserve_13 : BOOL ;
    reserve_14 : BOOL ;
    reserve_15 : BOOL ;
    res : BOOL ;
   END_STRUCT ;
   STATE : STRUCT
    Faulted : BOOL ;
    SETRECIPE_allowed : BOOL ;
    StopButtonAvalable : BOOL ;
    reserve_3 : BOOL ;
    reserve_4 : BOOL ;
    reserve_5 : BOOL ;
    reserve_6 : BOOL ;
    reserve_7 : BOOL ;
    reserve_8 : BOOL ;
    reserve_9 : BOOL ;
    reserve_10 : BOOL ;
    reserve_6_1 : BOOL ;
    reserve_7_1 : BOOL ;
    reserve_8_1 : BOOL ;
    reserve_9_1 : BOOL ;
    reserve_10_1 : BOOL ;
   END_STRUCT ;
   PARAM : STRUCT
    res_1 : REAL  := 2.000000e+000;
    res_2 : REAL  := 6.000000e+001;
    res_3 : REAL  := 6.000000e+001;
    MAN_RECIPENUMBER : INT ;
    reserve_4 : INT ;
    reserve_5 : INT ;
    reserve_6 : INT ;
    reserve_7 : INT ;
    reserve_8 : INT ;
    PressureCond : REAL  := -3.500000e+002;
    PulseValve : REAL  := 3.000000e+000;
    PauseValve : REAL  := 3.000000e+000;
    reserve_12 : REAL  := 1.000000e+001;
    reserve_13 : REAL  := 1.000000e+001;
   END_STRUCT ;
   PV : STRUCT
    res : REAL ;	//Minutes
    TON_HopperDischarge : REAL ;
    TON_RestDischarge : REAL ;
    res_2 : REAL ;
    reserve_1 : REAL ;
    StatusFilling : INT ;
    StatusDischarging : INT ;
    StatusHopper : INT ;
    res_3 : INT ;
    reserve_6 : INT ;
    RecipeNumber : INT ;
    RinneSpeed : REAL ;
    reserve_9 : REAL ;
    reserve_10 : REAL ;
    reserve_11 : REAL ;	//Minutes
   END_STRUCT ;
  END_STRUCT ;
  PROD : STRUCT 	//Interface of Production
   FROM : STRUCT
    reserve : INT ;
    reserve_1 : INT ;
    reserve_2 : INT ;
    reserve_3 : INT ;
    reserve_4 : INT ;
    reserve_5 : REAL ;
    reserve_6 : REAL ;
    CMD : STRUCT
     reserve : BOOL ;
     reserve_1 : BOOL ;
     reserve_2 : BOOL ;
     reserve_3 : BOOL ;
     reserve_4 : BOOL ;
     reserve_5 : BOOL ;
     reserve_6 : BOOL ;
     reserve_7 : BOOL ;
     reserve_8 : BOOL ;
     reserve_9 : BOOL ;
     reserve_10 : BOOL ;
     reserve_11 : BOOL ;
     reserve_12 : BOOL ;
     reserve_13 : BOOL ;
     reserve_14 : BOOL ;
     reserve_15 : BOOL ;
    END_STRUCT ;
   END_STRUCT ;
   TO : STRUCT
    reserve : INT ;
    reserve_1 : INT ;
    reserve_2 : INT ;
    reserve_3 : INT ;
    reserve_4 : INT ;
    reserve_5 : REAL ;
    reserve_6 : REAL ;
    STATE : STRUCT
     reserve : BOOL ;
     reserve_1 : BOOL ;
     reserve_2 : BOOL ;
     reserve_3 : BOOL ;
     reserve_4 : BOOL ;
     reserve_5 : BOOL ;
     reserve_6 : BOOL ;
     reserve_7 : BOOL ;
     reserve_8 : BOOL ;
     reserve_9 : BOOL ;
     reserve_10 : BOOL ;
     reserve_11 : BOOL ;
     reserve_12 : BOOL ;
     reserve_13 : BOOL ;
     reserve_14 : BOOL ;
     reserve_15 : BOOL ;
    END_STRUCT ;
   END_STRUCT ;
   reserve : ARRAY  [40 .. 49 ] OF BYTE ;
  END_STRUCT ;
  IF_RECEIVER : STRUCT 	//Interface scale in storage location
   CONTROL : STRUCT
    Answer_DB : INT ;
    Answer_DW : INT ;
    reserve : INT ;
    FrequencyRinne : INT ;
    RecipeNumber : INT ;
    ActualPressure : REAL ;
    reserve_4 : REAL ;
    CMD : STRUCT
     Connect : BOOL ;
     Request : BOOL ;
     Release : BOOL ;
     Full : BOOL ;
     CLEANING : BOOL ;
     PressureFault : BOOL ;
     SFStop : BOOL ;
     DISCH_SEQ_FAULT : BOOL ;
     DISCH_Agg_FAULT : BOOL ;
     FILL_SEQ_FAULT : BOOL ;
     FILL_Agg_FAULT : BOOL ;
     DischargingRECActive : BOOL ;
     AckMaterial : BOOL ;
     reserve_4 : BOOL ;
     reserve_5 : BOOL ;
     reserve_6 : BOOL ;
    END_STRUCT ;
   END_STRUCT ;
   STATUS : STRUCT
    reserve_1 : INT ;
    reserve_2 : INT ;
    reserve_3 : INT ;
    reserve_4 : INT ;
    RecipeNumber : INT ;
    reserve_6 : REAL ;
    reserve_7 : REAL ;
    STATE : STRUCT
     Ready : BOOL ;
     Active : BOOL ;
     RestDischarge : BOOL ;
     Faulted : BOOL ;
     HopperEmpty : BOOL ;
     HopperFilled : BOOL ;
     Stopped : BOOL ;
     TookRecipe : BOOL ;
     reserve_6 : BOOL ;
     reserve_7 : BOOL ;
     reserve_8 : BOOL ;
     reserve_9 : BOOL ;
     reserve_10 : BOOL ;
     reserve_11 : BOOL ;
     reserve_12 : BOOL ;
     reserve_13 : BOOL ;
    END_STRUCT ;
   END_STRUCT ;
  END_STRUCT ;
  reserve_IF : ARRAY  [236 .. 499 ] OF BYTE ;
  FAValve : STRUCT 	//valve object with 1Q and 0-2I
   parameter : STRUCT
    valve_on : BOOL  := TRUE;	//activate valve structure
    clock_on : BOOL ;	//activate clock structure
    reserve_3 : BOOL ;
    switching_number_on : BOOL ;	//activate switching number counter
    reserve_4 : BOOL ;
    parameter_1Q : BOOL ;	//valve type with 1 quit 0 inputs
    parameter_1Q_1I : BOOL ;	//valve type with 1 quit 1 input (=)
    parameter_1Q_1IN : BOOL ;	//valve type with 1 quit 1 input (<>)
    parameter_1Q_2I : BOOL  := TRUE;	//valve type with 1 quit 2 inputs
    parameter_text_pos_1 : BOOL ;
    parameter_text_straight : BOOL ;
    parameter_text_inverse : BOOL  := TRUE;	//select text inverse = "close/open" or "bypass/convey" aso.
    parameter_text_open : BOOL  := TRUE;	//select text quit = "open/close"
    parameter_text_convey : BOOL ;	//select text quit = "convey/bypass"
    parameter_text_on : BOOL ;	//select text quit = "on/off"
    parameter_text_up : BOOL ;	//select text quit = "up/down"
   END_STRUCT ;
   quit_valve : BOOL ;	//1 = quit valve
   input_valve_set : BOOL ;	//1 = input valve, if quit valve set
   input_valve_not_set : BOOL ;	//1 = input valve, if quit valve not set
   auto_mode_control : BOOL ;	//1 = release/control of valve in auto mode
   valve_in_operation : BOOL ;	//1 = signal valve in operation
   fault : BOOL ;	//1 = signal valve fault
   man_mode_to_SCADA : BOOL ;	//0 = automatic mode , 1 = manual mode
   man_mode_from_SCADA : BOOL ;	//0 = automatic mode , 1 = manual mode
   man_mode_control : BOOL ;	//1 = release/control of valve in manual mode (from SCADA)
   man_mode_locked : BOOL ;	//1 = change to manual mode locked, valve is in automatic use
   start_with_impulse : BOOL ;	//1 = start cycle with impluse
   set_cycles_reached : BOOL ;	//1 = set number of cycles has been reached
   continous_clock : BOOL ;	//1 = continous clock / 0 = set number of clocks
   simulation : BOOL ;	//1 = simulation of object
   release_clock : BOOL ;	//1 = release bit for clock FC
   quit_clock : BOOL ;	//quit for clock FC, if release_clock = TRUE
   set_time_fault : INT  := 5;	//fault evaluation time in seconds
   actual_time_fault : INT ;	//actual fault evaluation time in seconds
   impulse_time : REAL  := 5.000000e+000;	//impulse time for clock in seconds
   break_time : REAL  := 5.000000e+000;	//break time for clock in seconds
   time_counter : REAL ;	//time counter (elapsed time)
   set_cycles : INT ;	//number of clocks if not continous clock
   clock_counter : INT ;	//clock counter
   switching_number_counter : STRUCT 	//switching number counter
    reset : BOOL ;	//reset switching number counter
    warning : BOOL ;	//warning number exceeded
    alarm : BOOL ;	//alarm number exceeded
    flank_flag : BOOL ;	//internal flag
    actual_switching_number : REAL ;	//actual switching number
    set_number_warning : REAL ;	//set number for warning
    set_number_alarm : REAL ;	//set number for alarm
   END_STRUCT ;
   set_time_in_operation : INT ;	//1IoO: set time for delay of "valve in operation"
   real_time_in_operation : INT ;	//1IoO: real time for delay of "valve in operation"
   system_on : BOOL ;	//system released resepectively system area released after emergency stopping
   reserve : ARRAY  [44 .. 47 ] OF BYTE ;
   object_state : INT ;	//1=grey; 5=green; 9=white; 15=yellow; 16=red
  END_STRUCT ;
  reserve_Cmod_1 : ARRAY  [550 .. 799 ] OF BYTE ;
  BinaryObjects : STRUCT
   PBStart : STRUCT
    parameter : STRUCT
     reserve : BOOL ;
     debounce_time : BOOL ;	//view/edit debounce time
     reserve_2 : BOOL ;
     switching_number_counter : BOOL ;	//Counter for operating cycles
     reserve_4 : BOOL ;
     reserve_5 : BOOL ;
     reserve_6 : BOOL ;
     reserve_7 : BOOL ;
     parameter_invers : BOOL ;	//Parameter signal invers, invert the status
     reserve_9 : BOOL ;
     reserve_10 : BOOL ;
     reserve_11 : BOOL ;
     reserve_12 : BOOL ;
     reserve_13 : BOOL ;
     reserve_14 : BOOL ;
     reserve_15 : BOOL ;
    END_STRUCT ;
    input_processed : BOOL ;	//Input_signal processed
    input : BOOL ;	//Input signal
    def_invert_input : BOOL ;	//Definition to invert input signal (1=invert input)
    def_debounce_input : BOOL ;	//Definition to debounce input signal (1=debounce input)
    def_fault_state : BOOL ;	//Definition of fault state
    fault : BOOL ;	//1 = fault message
    man_mode_to_SCADA : BOOL ;	//0=Automode; 1=Manualmode
    man_mode_from_SCADA : BOOL ;	//0=Automode; 1=Manualmode
    man_mode_control : BOOL ;	//Control the object in manual mode (from scada)
    man_mode_locked : BOOL ;	//Lock manual mode, because object is used in auto mode
    system_on : BOOL ;
    spare : BOOL ;
    input_inverted : BOOL ;	//Input signal inverted if necessary
    input_debounced : BOOL ;	//Input signal debounced if necessary (also inverted if necessary9)
    input_debounced_high : BOOL ;	//Input signal debounced high (output signal timer)
    input_debounced_low : BOOL ;	//Input signal debounced low (output signal timer)
    set_time_fault : INT ;	//Set value fault evaulation time
    act_time_fault : INT ;	//Act value fault avaulation time
    set_time_debounced_high : REAL ;
    act_time_debounced_high : REAL ;
    set_time_debounced_low : REAL ;
    act_time_debounced_low : REAL ;
    cycle_counter : STRUCT
     reset_counter : BOOL ;	//Reset operating cycle counter
     warning : BOOL ;	//Warning time 1 elapsed
     alarm : BOOL ;	//Alarm time 2 elapsed
     flank_flag : BOOL ;	//Intern used flag
     act_number_of_cycles : REAL ;	//Actual number of cycles (cycle counter)
     set_number_warning : REAL ;	//Set value for generate the warning
     set_number_alarm : REAL ;	//Set value for generate the alarm
    END_STRUCT ;
    reserve : ARRAY  [38 .. 47 ] OF BYTE ;
    object_state : INT ;
   END_STRUCT ;
   PBStop : STRUCT
    parameter : STRUCT
     reserve : BOOL ;
     debounce_time : BOOL ;	//view/edit debounce time
     reserve_2 : BOOL ;
     switching_number_counter : BOOL ;	//Counter for operating cycles
     reserve_4 : BOOL ;
     reserve_5 : BOOL ;
     reserve_6 : BOOL ;
     reserve_7 : BOOL ;
     parameter_invers : BOOL ;	//Parameter signal invers, invert the status
     reserve_9 : BOOL ;
     reserve_10 : BOOL ;
     reserve_11 : BOOL ;
     reserve_12 : BOOL ;
     reserve_13 : BOOL ;
     reserve_14 : BOOL ;
     reserve_15 : BOOL ;
    END_STRUCT ;
    input_processed : BOOL ;	//Input_signal processed
    input : BOOL ;	//Input signal
    def_invert_input : BOOL ;	//Definition to invert input signal (1=invert input)
    def_debounce_input : BOOL ;	//Definition to debounce input signal (1=debounce input)
    def_fault_state : BOOL ;	//Definition of fault state
    fault : BOOL ;	//1 = fault message
    man_mode_to_SCADA : BOOL ;	//0=Automode; 1=Manualmode
    man_mode_from_SCADA : BOOL ;	//0=Automode; 1=Manualmode
    man_mode_control : BOOL ;	//Control the object in manual mode (from scada)
    man_mode_locked : BOOL ;	//Lock manual mode, because object is used in auto mode
    system_on : BOOL ;
    spare : BOOL ;
    input_inverted : BOOL ;	//Input signal inverted if necessary
    input_debounced : BOOL ;	//Input signal debounced if necessary (also inverted if necessary9)
    input_debounced_high : BOOL ;	//Input signal debounced high (output signal timer)
    input_debounced_low : BOOL ;	//Input signal debounced low (output signal timer)
    set_time_fault : INT ;	//Set value fault evaulation time
    act_time_fault : INT ;	//Act value fault avaulation time
    set_time_debounced_high : REAL ;
    act_time_debounced_high : REAL ;
    set_time_debounced_low : REAL ;
    act_time_debounced_low : REAL ;
    cycle_counter : STRUCT
     reset_counter : BOOL ;	//Reset operating cycle counter
     warning : BOOL ;	//Warning time 1 elapsed
     alarm : BOOL ;	//Alarm time 2 elapsed
     flank_flag : BOOL ;	//Intern used flag
     act_number_of_cycles : REAL ;	//Actual number of cycles (cycle counter)
     set_number_warning : REAL ;	//Set value for generate the warning
     set_number_alarm : REAL ;	//Set value for generate the alarm
    END_STRUCT ;
    reserve : ARRAY  [38 .. 47 ] OF BYTE ;
    object_state : INT ;
   END_STRUCT ;
   CstAvalible : STRUCT
    parameter : STRUCT
     reserve : BOOL ;
     debounce_time : BOOL ;	//view/edit debounce time
     reserve_2 : BOOL ;
     switching_number_counter : BOOL ;	//Counter for operating cycles
     reserve_4 : BOOL ;
     reserve_5 : BOOL ;
     reserve_6 : BOOL ;
     reserve_7 : BOOL ;
     parameter_invers : BOOL ;	//Parameter signal invers, invert the status
     reserve_9 : BOOL ;
     reserve_10 : BOOL ;
     reserve_11 : BOOL ;
     reserve_12 : BOOL ;
     reserve_13 : BOOL ;
     reserve_14 : BOOL ;
     reserve_15 : BOOL ;
    END_STRUCT ;
    input_processed : BOOL ;	//Input_signal processed
    input : BOOL ;	//Input signal
    def_invert_input : BOOL ;	//Definition to invert input signal (1=invert input)
    def_debounce_input : BOOL ;	//Definition to debounce input signal (1=debounce input)
    def_fault_state : BOOL ;	//Definition of fault state
    fault : BOOL ;	//1 = fault message
    man_mode_to_SCADA : BOOL ;	//0=Automode; 1=Manualmode
    man_mode_from_SCADA : BOOL ;	//0=Automode; 1=Manualmode
    man_mode_control : BOOL ;	//Control the object in manual mode (from scada)
    man_mode_locked : BOOL ;	//Lock manual mode, because object is used in auto mode
    system_on : BOOL ;
    spare : BOOL ;
    input_inverted : BOOL ;	//Input signal inverted if necessary
    input_debounced : BOOL ;	//Input signal debounced if necessary (also inverted if necessary9)
    input_debounced_high : BOOL ;	//Input signal debounced high (output signal timer)
    input_debounced_low : BOOL ;	//Input signal debounced low (output signal timer)
    set_time_fault : INT ;	//Set value fault evaulation time
    act_time_fault : INT ;	//Act value fault avaulation time
    set_time_debounced_high : REAL ;
    act_time_debounced_high : REAL ;
    set_time_debounced_low : REAL ;
    act_time_debounced_low : REAL ;
    cycle_counter : STRUCT
     reset_counter : BOOL ;	//Reset operating cycle counter
     warning : BOOL ;	//Warning time 1 elapsed
     alarm : BOOL ;	//Alarm time 2 elapsed
     flank_flag : BOOL ;	//Intern used flag
     act_number_of_cycles : REAL ;	//Actual number of cycles (cycle counter)
     set_number_warning : REAL ;	//Set value for generate the warning
     set_number_alarm : REAL ;	//Set value for generate the alarm
    END_STRUCT ;
    reserve : ARRAY  [38 .. 47 ] OF BYTE ;
    object_state : INT ;
   END_STRUCT ;
  END_STRUCT ;
  reserve_Cmod : ARRAY  [950 .. 1499 ] OF BYTE ;
  TIMES : STRUCT 	//ten timers
   TON_VibroRinneFault : STRUCT
    IN : BOOL ;
    RST : BOOL ;
    IMP : BOOL ;
    Q : BOOL ;
    PT : REAL ;
    ET : REAL ;
   END_STRUCT ;
   TON_Restdischarge : STRUCT
    IN : BOOL ;
    RST : BOOL ;
    IMP : BOOL ;
    Q : BOOL ;
    PT : REAL ;
    ET : REAL ;
   END_STRUCT ;
   TON_VibroRinneStart : STRUCT
    IN : BOOL ;
    RST : BOOL ;
    IMP : BOOL ;
    Q : BOOL ;
    PT : REAL ;
    ET : REAL ;
   END_STRUCT ;
   TON_HopperDischarge : STRUCT
    IN : BOOL ;
    RST : BOOL ;
    IMP : BOOL ;
    Q : BOOL ;
    PT : REAL ;
    ET : REAL ;
   END_STRUCT ;
   TON_Vibrorinne : STRUCT
    IN : BOOL ;
    RST : BOOL ;
    IMP : BOOL ;
    Q : BOOL ;
    PT : REAL ;
    ET : REAL ;
   END_STRUCT ;
  END_STRUCT ;
  SEQUENCES : STRUCT
   Filling : STRUCT
    AUTO : BOOL ;
    MANUAL : BOOL ;
    LOCKED : BOOL ;
    reserve : BOOL ;
    reserve_1 : BOOL ;
    reserve_2 : BOOL ;
    reserve_3 : BOOL ;
    reserve_4 : BOOL ;
    reserve_5 : BOOL ;
    reserve_6 : BOOL ;
    reserve_7 : BOOL ;
    reserve_8 : BOOL ;
    reserve_9 : BOOL ;
    reserve_10 : BOOL ;
    reserve_11 : BOOL ;
    reserve_12 : BOOL ;
   END_STRUCT ;
   Discharging : STRUCT
    AUTO : BOOL ;
    MANUAL : BOOL ;
    LOCKED : BOOL ;
    RELEASED : BOOL ;
    ACTIVE : BOOL ;
    HOPPERDISCHARGE : BOOL ;
    FAULTED : BOOL ;
    CLEANING : BOOL ;
    RESTDISCHARGE : BOOL ;
    reserve_5 : BOOL ;
    reserve_6 : BOOL ;
    reserve_7 : BOOL ;
    reserve_8 : BOOL ;
    reserve_9 : BOOL ;
    reserve_10 : BOOL ;
    reserve_11 : BOOL ;
   END_STRUCT ;
   reserve : ARRAY  [4 .. 99 ] OF BYTE ;
  END_STRUCT ;
  INTERNAL : STRUCT
   IF : STRUCT
    RECEIVER : STRUCT
     res : BOOL ;
     res_1 : BOOL ;
     res_2 : BOOL ;
     res_3 : BOOL ;
     res_4 : BOOL ;
     res_5 : BOOL ;
     res_6 : BOOL ;
     res_7 : BOOL ;
    END_STRUCT ;
    reserve_1 : BOOL ;
    reserve_2 : BOOL ;
    reserve_3 : BOOL ;
    reserve_4 : BOOL ;
    reserve_5 : BOOL ;
    reserve_6 : BOOL ;
    reserve_7 : BOOL ;
    reserve_8 : BOOL ;
    reserve_9 : BOOL ;
    reserve_10 : BOOL ;
    reserve_11 : BOOL ;
    reserve_12 : BOOL ;
    reserve_13 : BOOL ;
    reserve_14 : BOOL ;
    reserve_14_1 : BOOL ;
   END_STRUCT ;
   Flags : STRUCT
    FP_start : STRUCT
     helpbit : BOOL ;
     pulsebit : BOOL ;
    END_STRUCT ;
    xx_FP_FN : STRUCT
     helpbit : BOOL ;
     pulsebit : BOOL ;
    END_STRUCT ;
    FHP_Statuses : STRUCT
     HopperEmpty : BOOL ;
     HopperFilled : BOOL ;
     HopperDischargedFinished : BOOL ;
     RestDischargeFinished : BOOL ;
     res_1 : BOOL ;
     res_2 : BOOL ;
     res_3 : BOOL ;
     res_4 : BOOL ;
    END_STRUCT ;
    Switches : STRUCT
     res1 : BOOL ;
     res2 : BOOL ;
     res3 : BOOL ;
     res4 : BOOL ;
     res5 : BOOL ;
     res6 : BOOL ;
     res7 : BOOL ;
     ress8 : BOOL ;
     res9 : BOOL ;
     res10 : BOOL ;
     res11 : BOOL ;
    END_STRUCT ;
    BUTTONS_LAMPS : STRUCT
     LMStart : STRUCT
      Steady : BOOL ;
      Flash : BOOL ;
      DoubleFlash : BOOL ;
      Activated : BOOL ;
      res_1 : BOOL ;
      res_2 : BOOL ;
      res_3 : BOOL ;
      res_4 : BOOL ;
     END_STRUCT ;
     LMStop : STRUCT
      Steady : BOOL ;
      Flash : BOOL ;
      DoubleFlash : BOOL ;
      Activated : BOOL ;
      res_1 : BOOL ;
      res_2 : BOOL ;
      res_3 : BOOL ;
      res_4 : BOOL ;
     END_STRUCT ;
     LMCstAvalible : STRUCT
      Steady : BOOL ;
      Flash : BOOL ;
      DoubleFlash : BOOL ;
      Activated : BOOL ;
      res_1 : BOOL ;
      res_2 : BOOL ;
      res_3 : BOOL ;
      res_4 : BOOL ;
     END_STRUCT ;
     res_2_2 : BOOL ;
     res_3 : BOOL ;
     res_4 : BOOL ;
     res_5 : BOOL ;
     res_1_1 : BOOL ;
     res_2_1 : BOOL ;
     res_3_1 : BOOL ;
     res_4_1 : BOOL ;
     res_1 : BOOL ;
     res_2 : BOOL ;
    END_STRUCT ;
    BtnStartCMD : BOOL ;
    BtnStopCMD : BOOL ;
    extraPressureCondition : BOOL ;
    ValveExtraCond1 : BOOL ;
    ValveExtraCond2 : BOOL ;
    CstAvalible : BOOL ;
    res_2 : BOOL ;
    res_3 : BOOL ;
   END_STRUCT ;
   PARAM : STRUCT
    frequencyRinne : REAL ;
    res : REAL ;
    SpeedRinne : INT ;
   END_STRUCT ;
   Instance_DB_number : INT ;
  END_STRUCT ;
END_VAR
VAR_TEMP
  tempREAL : REAL ;
  tempINT : INT ;
  tempWORD : WORD ;
  tempBOOL : BOOL ;
END_VAR
BEGIN
NETWORK
TITLE = ------------------ INSTANCE DB (STANDART)-----------------------
      L     0;
      L     DINO;
      ==I;
      BEC;
      T     #INTERNAL.Instance_DB_number;
NETWORK
TITLE = -------------SEQUENCES AUTO/LOCKED/MANUAL-----------------
NETWORK
TITLE = Sequence discharging auto
      A     #IF_RECEIVER.CONTROL.CMD.Request;
      AN    #SEQUENCES.Discharging.LOCKED;
      =     #SEQUENCES.Discharging.AUTO;
NETWORK
TITLE = Sequence discharging manual
      O     #FAValve.man_mode_to_SCADA;
      AN    #SEQUENCES.Discharging.AUTO;
      =     #SEQUENCES.Discharging.MANUAL;
NETWORK
TITLE = Sequence discharging locked
      O     #SEQUENCES.Discharging.MANUAL;
      ON    #i_xSystemActive;
      =     #SEQUENCES.Discharging.LOCKED;
NETWORK
TITLE = ------------- SENSORS/SWITCHES/BINARY --------------------------
NETWORK
TITLE = LMP PBStart
      O     #i_xPBStart;
      O     #HMI.CMD.StartProd;
      =     #i_xPBStart;
      CALL  "FC24 Binär-E" (
           in_Handbedienung_erlaubt := TRUE,
           in_Anlage_ein            := #i_xSystemActive,
           in_Eingang               := #i_xPBStart,
           in_Eingang_drehen        := FALSE,
           in_Eingang_entprellen    := FALSE,
           in_Stoerauswertung_aktiv := FALSE,
           in_Quitt_Stoerung_noetig := FALSE,
           in_Stoer_Zustand         := FALSE,
           in_Quitt_Stoerung        := FALSE,
           io_Eingang_verarbeitet   := #INTERNAL.Flags.BUTTONS_LAMPS.LMStart.Activated,
           io_Stoerung              := #tempBOOL,
           io_Struktur              := #BinaryObjects.PBStart);
////////////////////////////////////////////////////////////////////////////////
NETWORK
TITLE = PB STOP
      O     #i_xPBStop;
      O     #HMI.CMD.StopProd;
      =     #i_xPBStop;
      CALL  "FC24 Binär-E" (
           in_Handbedienung_erlaubt := TRUE,
           in_Anlage_ein            := #i_xSystemActive,
           in_Eingang               := #i_xPBStop,
           in_Eingang_drehen        := FALSE,
           in_Eingang_entprellen    := FALSE,
           in_Stoerauswertung_aktiv := FALSE,
           in_Quitt_Stoerung_noetig := FALSE,
           in_Stoer_Zustand         := FALSE,
           in_Quitt_Stoerung        := FALSE,
           io_Eingang_verarbeitet   := #INTERNAL.Flags.BUTTONS_LAMPS.LMCstAvalible.Activated,
           io_Stoerung              := #tempBOOL,
           io_Struktur              := #BinaryObjects.PBStop);
NETWORK
TITLE = Lmp PB CST Avalible
      O     #i_xCstAvalible;
      O     #HMI.CMD.StartProd;
      =     #i_xPBStart;
      CALL  "FC24 Binär-E" (
           in_Handbedienung_erlaubt := TRUE,
           in_Anlage_ein            := #i_xSystemActive,
           in_Eingang               := #i_xCstAvalible,
           in_Eingang_drehen        := FALSE,
           in_Eingang_entprellen    := FALSE,
           in_Stoerauswertung_aktiv := FALSE,
           in_Quitt_Stoerung_noetig := FALSE,
           in_Stoer_Zustand         := FALSE,
           in_Quitt_Stoerung        := FALSE,
           io_Eingang_verarbeitet   := #INTERNAL.Flags.BUTTONS_LAMPS.LMCstAvalible.Activated,
           io_Stoerung              := #tempBOOL,
           io_Struktur              := #BinaryObjects.CstAvalible);
////////////////////////////////////////////////////////////////////////////////
NETWORK
TITLE = ------------SEQUENCES/HANDSHAKES DISCHARGING -----------
NETWORK
TITLE = Start Comd with "start" button
//Discussion - with Start/Stop buttons or from Panel
      A     #i_xSystemActive;
      A     #i_xPBStart;
      A     #INTERNAL.Flags.BUTTONS_LAMPS.LMStart.Activated;
      A     #IF_RECEIVER.CONTROL.CMD.Request;
      A     #SEQUENCES.Discharging.AUTO;
      FP    #INTERNAL.Flags.FP_start.helpbit;
      =     #INTERNAL.Flags.FP_start.pulsebit;
      A     #INTERNAL.Flags.FP_start.pulsebit;
      S     #INTERNAL.Flags.BtnStartCMD;
      ON    #i_xSystemActive;
      O     #i_xPBStop;
      O     #INTERNAL.Flags.BUTTONS_LAMPS.LMStop.Activated;
      R     #INTERNAL.Flags.BtnStartCMD;
      S     #INTERNAL.Flags.BtnStopCMD;
      O     #INTERNAL.Flags.BtnStartCMD;
      ON    #IF_RECEIVER.CONTROL.CMD.Request;
      R     #INTERNAL.Flags.BtnStopCMD;
NETWORK
TITLE = Discharging: FAULT SEQ
      O     #f_xFAValve;
      =     #SEQUENCES.Discharging.FAULTED;
NETWORK
TITLE = Discharging: RELEASE from REC01/ RELEASED SEQ
      A     #IF_RECEIVER.CONTROL.CMD.Release;
      AN    #IF_RECEIVER.CONTROL.CMD.Full;
      =     #SEQUENCES.Discharging.RELEASED;
NETWORK
TITLE = Discharge: ACTIVE SEQ
      A     #SEQUENCES.Discharging.RELEASED;
      A(;
      O     #FAValve.valve_in_operation;
      );
      =     #SEQUENCES.Discharging.ACTIVE;
NETWORK
TITLE = Discharge: CLEANING SEQ
      A     #IF_RECEIVER.CONTROL.CMD.CLEANING;
      =     #SEQUENCES.Discharging.CLEANING;
NETWORK
TITLE = Discharging: READY TO REC01
      A     #SEQUENCES.Discharging.AUTO;
      A(;
//>>test1
      A     #INTERNAL.Flags.BtnStartCMD;
      O;
      A     #SEQUENCES.Discharging.HOPPERDISCHARGE;
      O;
      A     #SEQUENCES.Discharging.RESTDISCHARGE;
//>>test1
//  O     
//      A     #INTERNAL.Flags.BtnStopCMD
//      AN    #INTERNAL.Flags.FHP_Statuses.HopperDischargedFinished
//      A     #INTERNAL.Flags.Switches.LowLevelProceeded
//      O     
//      A     #INTERNAL.Flags.BtnStopCMD
//      AN    #INTERNAL.Flags.FHP_Statuses.RestDischargeFinished
//      AN    #INTERNAL.Flags.Switches.LowLevelProceeded
      );
      A     #IF_RECEIVER.CONTROL.CMD.Request;
      =     #IF_RECEIVER.STATUS.STATE.Ready;
NETWORK
TITLE = Discharging: ACTIVE TO REC01
      A     #IF_RECEIVER.CONTROL.CMD.Release;
      A(;
      O     #INTERNAL.Flags.BtnStartCMD;
      O     #SEQUENCES.Discharging.HOPPERDISCHARGE;
      );
// O     #Magnet.auto_mode_control
      =     #IF_RECEIVER.STATUS.STATE.Active;
NETWORK
TITLE = Discharging: Recipe exchange
//    A     #IF_RECEIVER.CONTROL.CMD.Request  // //(001)
//      O     
      A     #IF_RECEIVER.CONTROL.CMD.Connect;
      A(;
      L     #IF_RECEIVER.CONTROL.RecipeNumber;
      L     #HMI.PV.RecipeNumber;
      ==I;
      );
      O;
      A     #INTERNAL.Flags.FHP_Statuses.HopperEmpty;
      O;
      A     #IF_RECEIVER.CONTROL.CMD.AckMaterial;
      JCN   LR;
      L     #IF_RECEIVER.CONTROL.RecipeNumber;
      T     #HMI.PV.RecipeNumber;
LR:   T     #IF_RECEIVER.STATUS.RecipeNumber;
      AN    #IF_RECEIVER.CONTROL.CMD.Request;
      AN    #SEQUENCES.Discharging.RELEASED;
      AN    #SEQUENCES.Discharging.ACTIVE;
      AN    #SEQUENCES.Discharging.HOPPERDISCHARGE;
      AN    #SEQUENCES.Discharging.CLEANING;
      AN    #SEQUENCES.Discharging.RESTDISCHARGE;
      AN    #INTERNAL.Flags.FHP_Statuses.HopperEmpty;
      =     #HMI.STATE.SETRECIPE_allowed;
NETWORK
TITLE = Discharging: Stop to REC
      A     #INTERNAL.Flags.BtnStopCMD;
      A(;
      A     #INTERNAL.Flags.FHP_Statuses.HopperDischargedFinished;
      A     #INTERNAL.Flags.Switches.res7;
      O;
      A     #INTERNAL.Flags.FHP_Statuses.RestDischargeFinished;
      AN    #INTERNAL.Flags.Switches.res7;
      O;
      AN    #SEQUENCES.Discharging.ACTIVE;
      AN    #SEQUENCES.Discharging.HOPPERDISCHARGE;
      AN    #SEQUENCES.Discharging.RESTDISCHARGE;
      AN    #SEQUENCES.Discharging.RELEASED;
      A     #INTERNAL.Flags.FHP_Statuses.HopperEmpty;
      );
      =     #IF_RECEIVER.STATUS.STATE.Stopped;
NETWORK
TITLE = --------------------HOPPER STATES-------------------------------
NETWORK
TITLE = ----------------RELEASES TO AGGREGATES-----------------------
NETWORK
TITLE = Discharging: Extra Condition for unload valve
//(001)
      A(;
      L     #IF_RECEIVER.CONTROL.ActualPressure;
      L     #HMI.PARAM.PressureCond;
      <R;
      );
      =     #INTERNAL.Flags.ValveExtraCond1;
NETWORK
TITLE = Discharging: Release Unload Valve
// (001) introduced on the comissioning
      A     #INTERNAL.Flags.ValveExtraCond1;
      O     #SEQUENCES.Discharging.CLEANING;
      JC    VPP1;	// valve pulse pause
      SET;
      R     #FAValve.continous_clock;
      R     #FAValve.release_clock;
      JU    VPP2;
VPP1: NOP   0;
      =     #FAValve.continous_clock;
      =     #FAValve.release_clock;
      L     #HMI.PARAM.PulseValve;
      T     #FAValve.impulse_time;
      L     #HMI.PARAM.PauseValve;
      T     #FAValve.break_time;
VPP2: NOP   0;
      A     #SEQUENCES.Discharging.AUTO;
      A(;
      O     #SEQUENCES.Discharging.RELEASED;
      O     #SEQUENCES.Discharging.HOPPERDISCHARGE;
      O     #SEQUENCES.Discharging.CLEANING;	// (001)
      );
//      AN    #SEQUENCES.Discharging.CLEANING          // //(001)
      AN    #IF_RECEIVER.CONTROL.CMD.PressureFault;
//     AN    #INTERNAL.Flags.ValveExtraCond2
      =     #FAValve.auto_mode_control;
// man mode locked
      A     #FAValve.auto_mode_control;
      AN    "Service Mode ExpertMode";
      =     #FAValve.man_mode_locked;
      CALL  "FC21 Ventil 1A0-2E" (
           in_Ventil_Typ            := 1,
           in_Handbedienung_erlaubt := "Release Man Mode Valves",
           in_Quitt_Stoerung_noetig := "AckObligatoryValves",
           in_Quitt_Stoerung        := #ack_FAValve,
           in_Anlage_ein            := #i_xSystemActive,
           in_Ansteuerung_Ventil    := #FAValve.auto_mode_control,
           in_Eingang_angesteuert   := #i_xFAValveOpen,
           in_Eingang_nicht_angest  := #i_xFAValveClosed,
           io_Ausgang_Ventil        := #q_xFAValve,
           io_Ventil_in_Betrieb     := #FAValve.valve_in_operation,
           io_Stoerung              := #FAValve.fault,
           io_Ventilstruktur        := #FAValve);
NETWORK
TITLE = -------------------STATUSES TO VISU-----------------------------
NETWORK
TITLE = Statuses SEQUENCES
//faulted
      A     #SEQUENCES.Discharging.FAULTED;
      =     #HMI.STATE.Faulted;
      AN    #SEQUENCES.Discharging.RELEASED;
      AN    #SEQUENCES.Discharging.ACTIVE;
      AN    #SEQUENCES.Discharging.HOPPERDISCHARGE;
      JCN   DRA;	// status release assignment
      L     0;
      JU    DAF;	// status assignmnet is finished 
DRA:  A     #SEQUENCES.Discharging.RELEASED;	//released
      AN    #SEQUENCES.Discharging.ACTIVE;
      AN    #SEQUENCES.Discharging.HOPPERDISCHARGE;
      JCN   DAA;	// status active 
      L     1;
      JU    DAF;
DAA:  A     #SEQUENCES.Discharging.RELEASED;	//active
      A     #SEQUENCES.Discharging.ACTIVE;
      AN    #SEQUENCES.Discharging.HOPPERDISCHARGE;
      AN    #SEQUENCES.Discharging.RESTDISCHARGE;
      JCN   DAR1;
      L     2;
      JU    DAF;
DAR1: A     #SEQUENCES.Discharging.HOPPERDISCHARGE;	//rest discharge         rec01
      AN    #SEQUENCES.Discharging.RESTDISCHARGE;
      JCN   DAR2;
      L     5;
      JU    DAF;
DAR2: A     #SEQUENCES.Discharging.RESTDISCHARGE;	//rest discharge         rec01
      JCN   DAF;
      L     3;
      JU    DAF;
DAF:  T     #HMI.PV.StatusDischarging;
NETWORK
TITLE = Stop Button available
      A     #SEQUENCES.Discharging.ACTIVE;
      O     #IF_RECEIVER.CONTROL.CMD.Request;
      =     #HMI.STATE.StopButtonAvalable;
NETWORK
TITLE = ------------------------LAMPS-----------------------------------
NETWORK
TITLE = lamp PB Start
      A     #IF_RECEIVER.CONTROL.CMD.Request;
//    A     #INTERNAL.Flags.FHP_Statuses.HopperEmpty
      =     #INTERNAL.Flags.BUTTONS_LAMPS.LMStart.Flash;
      A     #SEQUENCES.Discharging.ACTIVE;
      AN    #IF_RECEIVER.CONTROL.CMD.Full;
      AN    #SEQUENCES.Discharging.FAULTED;
      AN    #SEQUENCES.Discharging.CLEANING;
      AN    #SEQUENCES.Discharging.RESTDISCHARGE;
      =     #INTERNAL.Flags.BUTTONS_LAMPS.LMStart.Steady;
      A     #IF_RECEIVER.CONTROL.CMD.Full;
      =     #INTERNAL.Flags.BUTTONS_LAMPS.LMStart.DoubleFlash;
      CALL  "FC25 Lamp" (
           Steady                   := #INTERNAL.Flags.BUTTONS_LAMPS.LMStart.Steady,
           Flash                    := #INTERNAL.Flags.BUTTONS_LAMPS.LMStart.Flash,
           DoubleFlash              := #INTERNAL.Flags.BUTTONS_LAMPS.LMStart.DoubleFlash,
           LampTest                 := "GlobalLampTesting",
           Lamp                     := #q_xLMStart);
NETWORK
TITLE = lamp PB Cst Avalible
      CLR;
//    =     #INTERNAL.Flags.BUTTONS_LAMPS.PBCstAvalible.Steady
//    A     #IF_RECEIVER.CONTROL.CMD.DischargingRECActive
//      =     #INTERNAL.Flags.BUTTONS_LAMPS.PBCstAvalible.Flash
//   A     #SEQUENCES.Discharging.HOPPERDISCHARGE
      O     #SEQUENCES.Discharging.CLEANING;
      =     #INTERNAL.Flags.BUTTONS_LAMPS.LMCstAvalible.Flash;
      CALL  "FC25 Lamp" (
           Steady                   := #INTERNAL.Flags.BUTTONS_LAMPS.LMCstAvalible.Steady,
           Flash                    := #INTERNAL.Flags.BUTTONS_LAMPS.LMCstAvalible.Flash,
           DoubleFlash              := #INTERNAL.Flags.BUTTONS_LAMPS.LMCstAvalible.DoubleFlash,
           LampTest                 := "GlobalLampTesting",
           Lamp                     := #q_xLMCstAvalible);
NETWORK
TITLE = ----------------------INTERFACES-------------------------------
NETWORK
TITLE = Receiver
      CALL  "FC41 copy Obj-SST Slave" (
           i_SST_von_Ziel           := #IF_RECEIVER.CONTROL,
           i_SST_an_Ziel            := #IF_RECEIVER.STATUS);
END_FUNCTION_BLOCK

